// TwinCAT 3 PLC project PlcProject
// ProgramVersion: 3.1.4026.10
// libraries:
//   Tc2_Standard, * (Beckhoff Automation GmbH)
//   Tc2_System, * (Beckhoff Automation GmbH)
//   Tc3_IotBase, * (Beckhoff Automation GmbH)
// project tree:
//   01_HiveMQ_MQTT/ HiveMQ_MQTT.TcPOU
//   / MAIN.TcPOU, PlcTask.TcTTO
// real-time tasks:
//   TASK PlcTask: cycle T#10ms, priority 20, ADS port 350

CONFIGURATION PlcProject
    RESOURCE PLC ON TwinCAT3
        TASK PlcTask(INTERVAL := T#10ms, PRIORITY := 20);
        PROGRAM MAIN WITH PlcTask : MAIN;
    END_RESOURCE
END_CONFIGURATION

// ---- MAIN.TcPOU
PROGRAM MAIN
VAR
	programIsRunning : USINT;
	
	hiveMQ_MQTT : HiveMQ_MQTT;
END_VAR

programIsRunning := programIsRunning + 1;

hiveMQ_MQTT();
// hiveMQ_MQTT.CyclicCode();

END_PROGRAM

// ---- 01_HiveMQ_MQTT/HiveMQ_MQTT.TcPOU
FUNCTION_BLOCK HiveMQ_MQTT
VAR
	asd : FB_IotMqttClient := (sHostName := '5a4bc4b2d7c240d58dfbffe85ec21b83.s1.eu.hivemq.cloud');
	connect : BOOL := TRUE;
END_VAR

// asd(
// 	sClientId:= , 
// 	sHostName:= , 
// 	nHostPort:= , 
// 	sTopicPrefix:= , 
// 	nKeepAlive:= , 
// 	sUserName:= , 
// 	sUserPassword:= , 
// 	stWill:= , 
// 	stTLS:= , 
// 	ipMessageQueue:= , 
// 	bError=> , 
// 	hrErrorCode=> , 
// 	eConnectionState=> , 
// 	bConnected=> );
	
asd.Execute(connect);

METHOD CyclicCode
VAR_INPUT
END_VAR
END_METHOD

END_FUNCTION_BLOCK
